FUNCTION_BLOCK TcoTask_DownCounter EXTENDS TcoTask
VAR
	_SetUpValue		:	LINT;
	_CounterValue	:	LINT := -1;
	_InvokeCounter	: LINT;
	_DoneCounter	: LINT;
END_VAR

IF(THIS^._taskState = eTaskState.Requested) THEN
	CounterValue := SetUpValue;
	_InvokeCounter := _InvokeCounter + 1; 
END_IF;

IF(Execute()) THEN
	_CounterValue := _CounterValue - 1;
	DoneWhen(_CounterValue <= 0);			
END_IF

IF(THIS^._taskState = eTaskState.Done) THEN
	_DoneCounter := _DoneCounter + 1; 
END_IF;

PROPERTY CounterValue : LINT
GET
CounterValue := _CounterValue;
END_GET
SET
_CounterValue := CounterValue;
END_SET
END_PROPERTY

PROPERTY InTheMiddle : BOOL
GET
InTheMiddle := ABS(_SetUpValue-2*_CounterValue)<1;
END_GET
END_PROPERTY

PROPERTY SetUpValue : LINT
GET
SetUpValue	:= _SetUpValue;
END_GET
SET
_SetUpValue	:= SetUpValue;
END_SET
END_PROPERTY

END_FUNCTION_BLOCK

(* stored: Version 1.1.0.1, ProductVersion 3.1.4024.6
   POU TcoTask_DownCounter: Id {4cc6a6a3-1908-42e8-a63d-b13f9bca8455}, SpecialFunc None
   Property CounterValue: Id {11c233ef-f10c-4793-a4c8-a74b32875746}
   Get Get: Id {cbcda9df-9163-4cc9-8004-844c6ace0811}
   Set Set: Id {49a1bf47-ebb4-4518-a5d3-4cb250439f8c}
   Property InTheMiddle: Id {b9b6785c-f994-4e8e-9069-839e42e2180c}
   Get Get: Id {26a24943-b129-4ad5-bd48-7a90c7f6118f}
   Property SetUpValue: Id {b6871c3b-f824-4f12-9054-94fca3a4d2f5}
   Get Get: Id {ba03a06a-10d4-43c4-aa89-2986a076017f}
   Set Set: Id {ce6b57da-e6aa-40a4-9cea-81f9f41d056d} *)
